// TIA Portal V16 export
// export: Created 2024-09-05T17:40:14.5861299Z, ExportSetting WithDefaults, DisplayName Totally Integrated Automation Portal, DisplayVersion V16 Update 6, DisplayName TIA Portal Version Control Interface, DisplayVersion V16 Update 2, DisplayName TIA Portal Openness, DisplayVersion V16 Update 6, DisplayName STEP 7 Professional, DisplayVersion V16 Update 6, DisplayName STEP 7 Safety, DisplayVersion V16, DisplayName WinCC Advanced, DisplayVersion V16 Update 6
TYPE "UDT_ProductionProgram"
// stored: IsFailsafeCompliant false
   STRUCT
      "Name" : String[50];
      CupformingParametersLeft { S7_SetPoint := 'True'} : "UDT_FittingParameters";
      CupformingParametersRight { S7_SetPoint := 'True'} : "UDT_FittingParameters";
      St1Insertion { S7_SetPoint := 'True'} : Array[1..20] of Bool;
      St1InsertionUsed : Array[1..20] of Bool;
      FaureciaNumber : String;
      FaureciaNumberStartChar : Int;
      FaureciaNumberLength : Int;
      MechanicalType : Int;
      Camera_program : Array[0..4] of USInt;
      Riveting_program_left : Array[0..2] of USInt;
      Riveting_program_right : Array[0..2] of USInt;
      Total_number_of_rivets_4 : Bool;
      NumberOfReadings : Int;
      Readings : Array[1..4] of "UDT_ProductionReadings";
   END_STRUCT;
END_TYPE
